Omron CX-Programmer project NewProject (CX-Programmer 9.75)

# PLC SubRoutine: CP1E N30

## Global symbols (name address type ; comment)
T000 BOOL  ; T0

## Program NewProgram1 (cyclic task 0)
Local symbols
AC 1.02 BOOL  ; 102
Fan 1.01 BOOL  ; 101
Light 100.03 BOOL  ; 100.3
Light2 100.07 BOOL  ; 100.07
Light3 100.09 BOOL  ; 100.09
M1 100.00 BOOL  ; 100.00
M2 100.01 BOOL  ; 100.01
M3 100.02 BOOL  ; 100.02
Motor1 1.03 BOOL  ; 103
Motor2 1.04 BOOL  ; 104
Start1 0.00 BOOL  ; 0.00
Start2 0.02 BOOL  ; 0.02
Start3 0.04 BOOL  ; 0.04
Stop1 0.01 BOOL  ; 0.01
Stop2 0.03 BOOL  ; 0.03
Stop3 0.05 BOOL  ; 0.05
Sw1 0.06 BOOL  ; 0.06
Sw3 0.07 BOOL  ; 0.07
Sw4 0.08 BOOL  ; 0.08
Switch2 1.00 BOOL  ; 1.00

### Section Control_panel

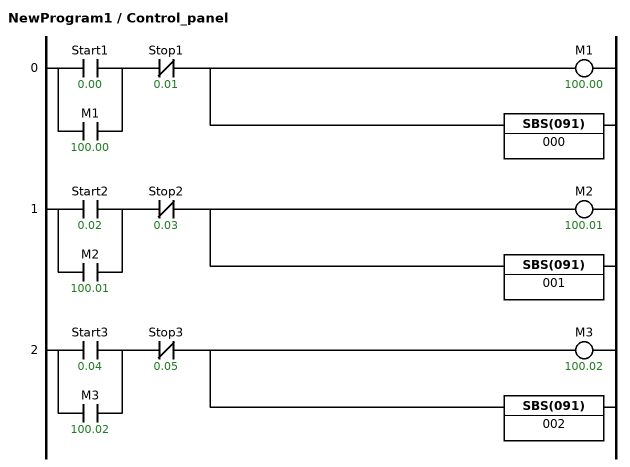
; rung 0
LD Start1  ; 0.00
OR M1  ; 100.00
ANDNOT Stop1  ; 0.01
OUT M1  ; 100.00
SBS(091) 000
; rung 1
LD Start2  ; 0.02
OR M2  ; 100.01
ANDNOT Stop2  ; 0.03
OUT M2  ; 100.01
SBS(091) 001
; rung 2
LD Start3  ; 0.04
OR M3  ; 100.02
ANDNOT Stop3  ; 0.05
OUT M3  ; 100.02
SBS(091) 002

### Section Phase_R

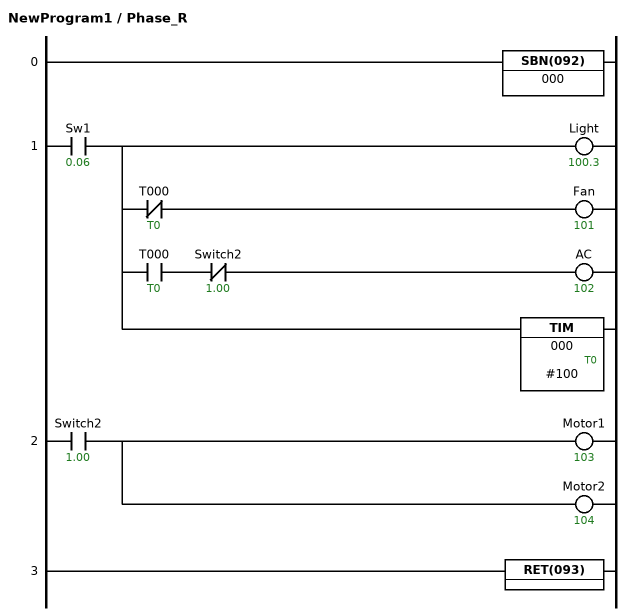
; rung 0
SBN(092) 000
; rung 1
LD Sw1  ; 0.06
OUT TR0
OUT Light  ; 100.3
ANDNOT T000  ; T0
OUT Fan  ; 101
LD TR0
AND T000  ; T0
ANDNOT Switch2  ; 1.00
OUT AC  ; 102
LD TR0
TIM 000 #100  ; T0
; rung 2
LD Switch2  ; 1.00
OUT Motor1  ; 103
OUT Motor2  ; 104
; rung 3
RET(093)

### Section Phase_Y

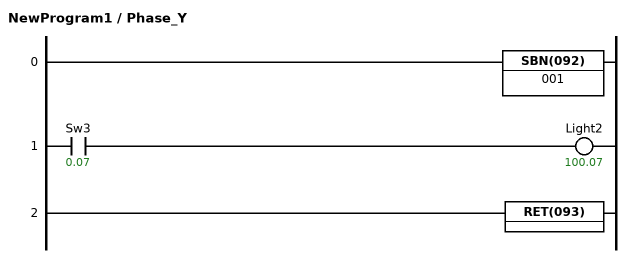
; rung 0
SBN(092) 001
; rung 1
LD Sw3  ; 0.07
OUT Light2  ; 100.07
; rung 2
RET(093)

### Section Phase_B

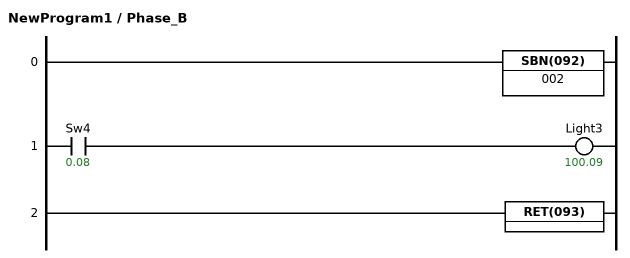
; rung 0
SBN(092) 002
; rung 1
LD Sw4  ; 0.08
OUT Light3  ; 100.09
; rung 2
RET(093)

### Section END
; rung 0
END(001)